PROGRAM PRG_UpdatePressureSensor
VAR
	evtPressureControlStart		: DetectEvent;
	evtPressureControlStop		: DetectEvent;
	
END_VAR

(* convert the pressure signal *)
pressureBar := INT_TO_REAL(pressureRawCounts)*pressureSensorCalibration.scaleFactor + pressureSensorCalibration.offset;


(* button events *)
evtPressureControlStart(newSignalValue := pressureStart);
evtPressureControlStop(newSignalValue := pressureStop);

IF evtPressureControlStart.eventDetected = TASTEVT_PositiveEdge THEN
	pressureStart := FALSE;
	pressureRunning := TRUE;
END_IF

IF evtPressureControlStop.eventDetected = TASTEVT_PositiveEdge THEN
	pressureStop := FALSE;
	pressureRunning := FALSE;
END_IF


(* controller *)
IF pressureRunning THEN
	IF pressureBar > pressureSetBar + 0.01  THEN
		reactorPressureInletValve := FALSE;
	END_IF
	
	IF pressureBar < pressureSetBar - 0.01 THEN
		reactorPressureInletValve := TRUE;
	END_IF
ELSE
	reactorPressureInletValve := FALSE;
END_IF

END_PROGRAM

(* stored: Version 1.1.0.1, ProductVersion 3.1.4022.7
   POU PRG_UpdatePressureSensor: Id {627c2f6a-4707-48e2-9348-f660345fe98d}, SpecialFunc None *)
